(* PLC project 05_drive_oop.project, CODESYS CODESYS V3.5 SP22 Patch 3 *)
(* stored: creationDateTime 2026-09-17T21:27:57.3785581, modificationDateTime 2026-09-17T21:27:15.8308055 *)

{attribute 'qualified_only'}
{attribute 'strict'}
TYPE E_DriveState : (IDLE := 0, RUNNING := 10, FAULT := 99);
END_TYPE

TYPE ST_Drive : STRUCT
  sName : STRING(20);
  rSpeedSet : REAL := 0.0;
  aCurrent : ARRAY[1..3] OF REAL;
  eState : E_DriveState := E_DriveState.IDLE;
END_STRUCT;
END_TYPE

PROGRAM PLC_PRG
  VAR
    fbDrive : FB_Drive;
    xStart : BOOL;
    xOk : BOOL;
    rActual : REAL;
  END_VAR

                    fbDrive(xEnable := TRUE);
IF xStart THEN
    xOk := fbDrive.M_Start(rTarget := 1500.0);
    xStart := FALSE;
END_IF
fbDrive.P_Speed := 1200.0;
rActual := fbDrive.P_Speed;
IF NOT fbDrive.xRunning THEN
    fbDrive.A_Reset();
END_IF
                  
END_PROGRAM

FUNCTION_BLOCK FB_Drive
  VAR_INPUT
    xEnable : BOOL;
  END_VAR
  VAR_OUTPUT
    xRunning : BOOL;
  END_VAR
  VAR
    stData : ST_Drive;
    rSpeed : REAL;
  END_VAR

                    xRunning := xEnable AND (stData.eState = E_DriveState.RUNNING);
                  

ACTION A_Reset:
                        stData.eState := E_DriveState.IDLE;
stData.rSpeedSet := 0.0;
                      
END_ACTION

METHOD M_Start : BOOL
  VAR_INPUT
    rTarget : REAL;
  END_VAR
  VAR
    xOk : BOOL;
  END_VAR
                          xOk := rTarget >= 0.0;
IF xOk THEN
    stData.rSpeedSet := rTarget;
    stData.eState := E_DriveState.RUNNING;
END_IF
M_Start := xOk;
                        
END_METHOD

PROPERTY P_Speed : REAL
GET
                             P_Speed := rSpeed;
                          
END_GET
SET
                            rSpeed := P_Speed;
                          
END_SET
END_PROPERTY
END_FUNCTION_BLOCK

CONFIGURATION Device
  RESOURCE Application ON PLC
    TASK MainTask(INTERVAL := T#20ms, PRIORITY := 1);
    PROGRAM PLC_PRG WITH MainTask : PLC_PRG;
  END_RESOURCE
END_CONFIGURATION
